Staubli VAL3: page_viewPallet.dtx

num nIndex
num nKey
num nMax
num nRefresh
num nTime = 2
num nView
string sEvent
public string sItems
string sList
string sMenu
string sMessage
string sPalletName
bool bButton[8]
bool bLarge
bool bOnActionLine
frame fView = {fatherId=world[0]}
pointRx pOrigin = {wrist=wfree, fatherId=fView[0]}
pointRx pPoints[4]
  [0] = {wrist=wfree, fatherId=world[0]}
  [1] = {wrist=wfree, fatherId=world[0]}
  [2] = {wrist=wfree, fatherId=world[0]}
  [3] = {wrist=wfree, fatherId=world[0]}
